// TIA Portal V18 export
DATA_BLOCK "idbMoteurAsynchrone"   // DB5
// stored: InstanceOfName nsConvoyeur.fbMoteurAsynchrone, InstanceOfType FB, Namespace nsConvoyeur
"nsConvoyeur.fbMoteurAsynchrone"
   // VAR_INPUT
   //    "iStart/Stop" : Bool;
   //    iAccelerate : Bool;
   //    iDecelerate : Bool;
   // END_VAR
   // VAR_IN_OUT
   //    ioPosition : UDInt;
   // END_VAR
BEGIN
END_DATA_BLOCK
